Fanuc KAREL source: kb00061.KL

-- PROVISIONAL review KL for V770-1; original PC SHA256 24fd546f0b1bbb3b4cd9db82f2148994a2e6e7d9d7dacb12926b9bf803ca776a
-- Incomplete behavior may be omitted. Consult companion uncertainty JSON. Do not deploy.
PROGRAM KB00061
%NOLOCKGROUP
BEGIN
  -- UNRESOLVED_PC offsets 5-14; opcodes 3F,75
  -- UNRESOLVED_PC offsets 19-26; opcodes 9D,23
  -- UNRESOLVED_PC offsets 31-38; opcodes 9D,23
  -- UNRESOLVED_PC offsets 43-67; opcodes 27,22,2A,22,22,31
  -- UNRESOLVED_PC offsets 72-76; opcodes 7F
END KB00061
